FUNCTION_BLOCK FB_Observable_DWORD EXTENDS FB_AbstractObservable
VAR
    _nVal:              DWORD;
    _nOldVal:           DWORD;
END_VAR

METHOD FB_init : BOOL
VAR_INPUT
    bInitRetains:       BOOL; // if TRUE, the retain variables are initialized (warm start / cold start)
    bInCopyCode:        BOOL;  // if TRUE, the instance afterwards gets moved into the copy code (online change)
END_VAR
THIS^._nTypeClass := __SYSTEM.TYPE_CLASS.TYPE_DWORD;
END_METHOD

PROPERTY nDataSize : UDINT
GET
nDataSize := SIZEOF(DWORD);
END_GET
END_PROPERTY

PROPERTY nValue32 : DWORD
GET
nValue32 := THIS^._nVal;
END_GET
SET
THIS^._nOldVal := THIS^._nVal;
THIS^._nVal := nValue32;

THIS^.NotifyWithConditions();
END_SET
END_PROPERTY

PROPERTY PROTECTED pData : POINTER TO BYTE
GET
pData := ADR(THIS^._nVal);
END_GET
END_PROPERTY

METHOD  ValueChanged : BOOL
VAR_INPUT
END_VAR
ValueChanged := THIS^._nOldVal <> THIS^._nVal;
END_METHOD

END_FUNCTION_BLOCK

(* stored: Version 1.1.0.1, ProductVersion 3.1.4024.12
   POU FB_Observable_DWORD: Id {7927e7e0-31c0-0121-269a-d66cae2acc85}, SpecialFunc None
   Method FB_init: Id {c9866173-54aa-09cb-3091-06d6dbfa477a}
   Property nDataSize: Id {9a7fa283-2e7f-00d5-1038-a29e74f126f4}
   Get Get: Id {47efd5ce-7bc7-0956-011a-fa12c5c2e844}
   Property nValue32: Id {a495e55a-2422-0bce-3cc1-0f416a7f561f}
   Get Get: Id {d6a18b5e-4bbe-0242-0fde-fd2b1cd86a14}
   Set Set: Id {316f1d94-6fca-08cd-0be0-98e321570525}
   Property pData: Id {8ed2da57-0387-0e62-3443-46e7c228416d}
   Get Get: Id {2313a11b-9ce5-00c1-31b2-46ef256b26c1}
   Method ValueChanged: Id {35b8b5b7-3a80-05b3-15e7-e9f02ba0d4f3} *)
